(*
Short description of the function.

Long description of the function, spanning multiple
rows even.
*)
FUNCTION RegularFunction : LREAL
VAR_INPUT
    input       : LREAL;            // This is an in-code description of some variable
    other_arg   : UDINT;
END_VAR
VAR
END_VAR

RegularFunction := input * 2.0;

END_FUNCTION

(* stored: Version 1.1.0.1, ProductVersion 3.1.4024.11
   POU RegularFunction: Id {f80a8020-3966-4dae-a6c7-7aceb360dfeb}, SpecialFunc None *)
